// TIA Portal V19 export
TYPE "CTRL_DIN"
   STRUCT
      status : Bool;
      sim : "UDT_SIM_BOOL";
   END_STRUCT;
END_TYPE
